FUNCTION_BLOCK FB_MachineModeSwitch EXTENDS FB_ObjectBase_V2
VAR_INPUT
	ModeLink 				 : REFERENCE TO ST_Mode;
	MachineCtrl_CurrentMode  : E_UnitMode;
	MachineCtrl_CurrentState : E_PMLState;
	MachineHomed			 : BOOL;
END_VAR
VAR_OUTPUT
	RequestedMode		 : E_UnitMode;
	ModeRequestValid	 : BOOL;
END_VAR
VAR
	eTargetModeCache    : E_MachineMode;

	eActualModeCache    : E_UnitMode;

	strStatus           : STRING;
	_bRetry				: BOOL;
	uiResumeStep		: UDINT;
	
	TON_WaitModeSwitch	: TON;
END_VAR

THIS^.A00_BasicUnits();
SUPER^.A10_StateControl();

IF PackTags[0].Status.UnitModeCurrent = E_UnitMode.Manual THEN
	GVL_ADS.MachineMode.CurrentMode := E_MachineMode.MANUAL;
ELSIF PackTags[0].Status.UnitModeCurrent = E_UnitMode.Auto THEN
	GVL_ADS.MachineMode.CurrentMode := E_MachineMode.AUTO;
END_IF

ACTION A00_BasicUnits:
eTargetModeCache := ModeLink.TargetMode;

eActualModeCache := GVL_Machine.PackTags[0].Status.UnitModeCurrent;

TON_WaitModeSwitch(PT := T#3S);
END_ACTION

METHOD M_CheckCommand : BOOL
VAR_INPUT
END_VAR
IF eTargetModeCache = E_MachineMode.AUTO AND NOT MachineHomed THEN
	strStatus := 'FB_MachineModeSwitch ,Not Homing can not Switch AutoMode not can retry';
	M_CheckCommand:= FALSE;
	RETURN;
END_IF

M_CheckCommand := TRUE;
END_METHOD

METHOD  M_STATE_ABORTED
VAR_INPUT
END_VAR
IF NOT _bRetry THEN
	Busy 	:= FALSE;
	Aborted := TRUE;
	Error 	:= TRUE;
	Status 	:= strStatus;
	uiAbortingStep := 0;
	_AbortCompleted := FALSE;
END_IF

IF reset THEN
	_bRetry := TRUE;
	Error	:= FALSE;
	Aborted	:= FALSE;
END_IF

IF NOT Execute THEN
	eState := STATE_RESETTING;
ELSIF Execute AND _bRetry THEN
	uiExecutingStep := uiResumeStep ;
	status :='';
	eState := STATE_EXECUTING;
END_IF
END_METHOD

METHOD  M_STATE_ABORTING
VAR_INPUT
END_VAR
Busy := FALSE;
Done := FALSE;
Aborted := FALSE;
Error := FALSE;
Status := strStatus;

CASE uiAbortingStep OF
	0:
		ModeRequestValid := FALSE;
		TON_WaitModeSwitch.IN := FALSE;
		_Abort := FALSE;
		_bRetry := FALSE;

		uiAbortingStep := 9999;

	9999:
		_AbortCompleted := TRUE;
END_CASE

IF _AbortCompleted THEN
	eState := STATE_ABORTED;
END_IF
END_METHOD

METHOD  M_STATE_DONE
VAR_INPUT
END_VAR
Busy := FALSE;
Done := TRUE;
Aborted := FALSE;
Error := FALSE;
Status := strStatus;

IF Reset OR NOT Execute THEN
	eState := STATE_RESETTING;
END_IF
END_METHOD

METHOD  M_STATE_DORMANT
VAR_INPUT
END_VAR
Busy := FALSE;
Done := FALSE;
Aborted := FALSE;
Error := FALSE;
Paused := FALSE;
Status := '';
UniqueErrorCode := '';

_Executed := FALSE;
_Error := FALSE;
_Abort := FALSE;
_ResetCompleted := FALSE;
_AbortCompleted := FALSE;
_HoldingCompleted := FALSE;
_HeldCompleted := FALSE;
_UnholdCompleted := FALSE;

uiExecutingStep := 0;
uiResettingStep := 0;
uiAbortingStep 	:= 0;
uiHoldingStep 	:= 0;
uiHeldStep 		:= 0;
uiUnholdStep 	:= 0;
uiResumeStep 	:= 0;

_bRetry := FALSE;
TON_WaitModeSwitch.IN := FALSE;
ModeRequestValid := FALSE;

strStatus := 'Machine mode switch idle';
Status := strStatus;

IF Execute THEN
	eState := STATE_EXECUTING;
END_IF
END_METHOD

METHOD  M_STATE_ERROR
VAR_INPUT
END_VAR
Busy := FALSE;
Error := TRUE;
Status := strStatus;
ModeRequestValid := FALSE;

IF NOT Execute THEN
	eState := STATE_RESETTING;
END_IF
END_METHOD

METHOD  M_STATE_EXECUTING
VAR_INPUT
END_VAR

VAR
	esle: INT;
END_VAR
Busy := TRUE;
Done := FALSE;
Aborted := FALSE;
Error := FALSE;

CASE uiExecutingStep OF
	0:
		IF M_CheckCommand() THEN
			uiExecutingStep := 100;
		ELSE
			_Error := TRUE;
		END_IF

	100:
		CASE eTargetModeCache OF
			E_MachineMode.MANUAL:
				TON_WaitModeSwitch.IN 	:= TRUE;
				RequestedMode 			:= E_UnitMode.Manual;
				ModeRequestValid 		:= TRUE;
				IF eActualModeCache = E_UnitMode.Manual THEN
					uiExecutingStep := 200;
				END_IF
				IF TON_WaitModeSwitch.Q THEN
					strStatus := 'FB_MachineModeSwitch ,Switch ManualMode Timeout';
					_Abort := TRUE;
				END_IF
				IF MachineCtrl_CurrentMode = E_UnitMode.Auto AND 
					MachineCtrl_CurrentState = E_PMLState.ePMLState_Suspended  THEN
					uiResumeStep := 100;
					strStatus 	 := 'FB_MachineModeSwitch ,MachineMode stuck in AutoMode Suspended , cat retry';
					_Abort    	 := TRUE;
				END_IF  

			E_MachineMode.AUTO:
				TON_WaitModeSwitch.IN 	:= TRUE;
				RequestedMode 			:= E_UnitMode.Auto;
				ModeRequestValid 		:= TRUE;
				IF eActualModeCache = E_UnitMode.Auto THEN
					uiExecutingStep := 200;
				END_IF
				IF TON_WaitModeSwitch.Q THEN
					strStatus := 'FB_MachineModeSwitch ,Switch AutoMode Timeout';
					_Abort := TRUE;
				END_IF
		ELSE
			ModeRequestValid := FALSE;
			strStatus := 'FB_MachineModeSwitch ,TargetMode is invalid for verification';
			_Error := TRUE;
		END_CASE

	200:
		ModeLink.CurrentMode := eTargetModeCache;
		
		strStatus := 'Machine mode switch verify complete';
		_Executed := TRUE;
END_CASE

IF NOT Execute THEN
	eState := STATE_RESETTING;
ELSIF _Error THEN
	eState := STATE_ERROR;
ELSIF _Abort THEN
	eState := STATE_ABORTING;
ELSIF _Executed THEN
	eState := STATE_DONE;
END_IF
END_METHOD

METHOD  M_STATE_RESETTING
VAR_INPUT
END_VAR
Busy := FALSE;
Aborted := FALSE;
Error := FALSE;

CASE uiResettingStep OF
	0:
		ModeRequestValid := FALSE;
		TON_WaitModeSwitch.IN := FALSE;

		uiResettingStep := 100;

	100:
		_ResetCompleted := TRUE;
END_CASE

IF _ResetCompleted THEN
	eState := STATE_DORMANT;
END_IF
END_METHOD

END_FUNCTION_BLOCK

(* stored: Version 1.1.0.1, ProductVersion 3.1.4024.13
   POU FB_MachineModeSwitch: Id {53c0ad14-faa3-42bf-b2f6-e8a0ec4c3d82}, SpecialFunc None
   Folder Method: Id {5f03531e-ec1c-469c-91db-8cd0961dc2bd}
   Folder STATE: Id {e593c19a-84fd-482a-a32d-e1e324d24f89}
   Action A00_BasicUnits: Id {a8e0054e-cc88-46e4-b0f7-533972befea0}
   Method M_CheckCommand: Id {5f3aac03-40f5-4913-b8ae-d7613f3e4f82}
   Method M_STATE_ABORTED: Id {b0cb5487-c094-4220-b311-09c79f325d32}
   Method M_STATE_ABORTING: Id {5101d1f1-ea45-4aef-9a7f-b770cfe9a43f}
   Method M_STATE_DONE: Id {7d1bfebf-6ba7-4f9e-ba18-bf103887b5b4}
   Method M_STATE_DORMANT: Id {c4b32cd1-cb28-42c0-8804-d1d35e09f97f}
   Method M_STATE_ERROR: Id {0689463d-acd2-484e-8eeb-7ff89d4312d2}
   Method M_STATE_EXECUTING: Id {80af41fd-0a13-4d38-aaf8-e19f9d81e0e7}
   Method M_STATE_RESETTING: Id {a34cb8a5-ee8d-4abd-ac41-e2995521a3c1} *)
